// 隐含生成代码：不要编辑
FUNCTION CheckDivReal : REAL
VAR_INPUT
	divisor:REAL;
END_VAR

// 隐含生成代码：这里只是对代码实现的建议
{noflow}
IF divisor = 0 THEN
	CheckDivReal:=1;
ELSE
	CheckDivReal:=divisor;
END_IF;
{flow}

END_FUNCTION

(* stored: Version 1.1.0.1, ProductVersion 3.1.4024.12
   POU CheckDivReal: Id {8b0d8229-7fb1-4359-92f8-2e2831f1d321}, SpecialFunc CheckDivReal32 *)
